(* Logix 5000 project; controller CLASE_1 Emulate 5570 rev 28.11; software revision 28.02; part 3 of 15 *)
(* tags used below, declared in another part *)
   Inp : BOOL;   // Alarm Condition Input 1=Alarm
   Cfg_Exists : BOOL;   // 1=Alarm configured to exist, 0=Does not exist, don't scan
   Cfg_ResetReqd : BOOL;   // 1=Latched Alarm, a Reset is required to clear this Alarm
   Cfg_AckReqd : BOOL;   // 1=Acknowledge required for this Alarm
   Cfg_AllowShelve : BOOL;   // 1=Allow Operator to Shelve this Alarm
   Cfg_AllowDisable : BOOL;   // 1=Allow Maintenance to Disable this Alarm
   Cfg_Severity : INT;   // Alarm Severity: 1..250=Low, 251..500=Medium, 501..750=High, 751..1000=Urgent
   Cfg_AlmMinOnT : DINT;   // Minimum time Alm output stays on (sec)
   Cfg_MaxShelfT : INT;   // Auto unshelve after shelved this long (1..32767 minutes)
   PCfg_AllowExist : BOOL;   // 1=Alarm can be configured to exist, 0=other configs make alarm meaningless
   PCmd_Ack : BOOL;   // Program Command to Acknowledge alarm
   PCmd_Suppress : BOOL;   // Program Command to Suppress by Design (inhibits new alarm)
   PCmd_Unsuppress : BOOL;   // Program Command to Unsuppress (allows new alarm)
   PCmd_Unshelve : BOOL;   // Program Command to Unshelve (e.g., on shift change)
   OCmd_Ack : BOOL;   // Operator Command to Acknowledge alarm
   OCmd_Shelve : BOOL;   // Operator Command to Shelve Alarm (inhibits new alarm)
   OCmd_Unshelve : BOOL;   // Operator Command to Unshelve alarm (allows new alarm)
   MCmd_Disable : BOOL;   // Maintenance Command to Disable alarm (inhibits new alarm)
   MCmd_Enable : BOOL;   // Maintenance Command to Enable alarm (allows new alarm)
   MCmd_Test : BOOL;   // Maintenance Command to Test alarm (issued for minimum alarm time)
   Val_MinToUnshelve : DINT;   // Number of minutes until this alarm unshelves itself (mmm:ss)
   Val_SecToUnshelve : DINT;   // Number of Seconds until this alarm unshelves itself (mmm:ss)
   Alm : ALIAS FOR Com_AE.0;   // Alarm output 1=In Alarm
   Ack : ALIAS FOR Com_AE.1;   // Alarm acknowledged status: 1=Ack rcvd
   Shelved : ALIAS FOR Com_AE.3;   // 1=Alarm has been Shelved by Operator (inhibits new alarm)
   Suppressed : ALIAS FOR Com_AE.6;   // 1=Alarm has been Suppressed by Program (inhibits new alarm)
   Disabled : ALIAS FOR Com_AE.9;   // 1=Alarm has been Disabled by Maintanance (inhibits new alarm)
   Err_Severity : BOOL;   // 1=Error in Config: Invalid Severity (use 1 to 4)
   Rdy_Ack : BOOL;   // Ready to receive OCmd_Ack (enables button)
   Rdy_Shelve : BOOL;   // Ready to receive OCmd_Shelve (enables button)
   Rdy_Unshelve : BOOL;   // Ready to receive OCmd_Unshelve (enables button)
   Rdy_Disable : BOOL;   // Ready to receive MCmd_Disable (enables button)
   Rdy_Enable : BOOL;   // Ready to receive MCmd_Enable (enables button)
   Rdy_Test : BOOL;   // Ready to receive MCmd_Test (enables button)
   P_Alarm : BOOL;   // Unique Parameter Name for auto - discovery
   Wrk_Alm : BOOL;   // Internal Alarm Status
   Wrk_Suppressed : BOOL;   // Internal Alarm Suppressed Status
   Wrk_AlmMinOnT : TIMER;   // Alarm output minimum ON time to be seen by alarm server
   Wrk_AutoAckT : TIMER;   // Time to clear Ack bit when Ack not required
   Wrk_ShelfT : TIMER;   // Time to auto Unshelve a Shelved Alarm
   Com_AE : INT;   // Communication with HMI / Alarm/Event Server (see bit descriptions)
   Cfg_Cond : STRING_20;   // Alarm Condition Text (e.g., "High-High PV")
   Wrk_SecToUnshelve : DINT;   // Number of seconds until this alarm unshelves itself
(* P_Alarm, continued *)

ROUTINE Logic   (* ladder *)
// Perform Alarm processing: delay, latch/reset, acknowledge, enable/disable, inhibit/uninhibit, suppress/unsuppress
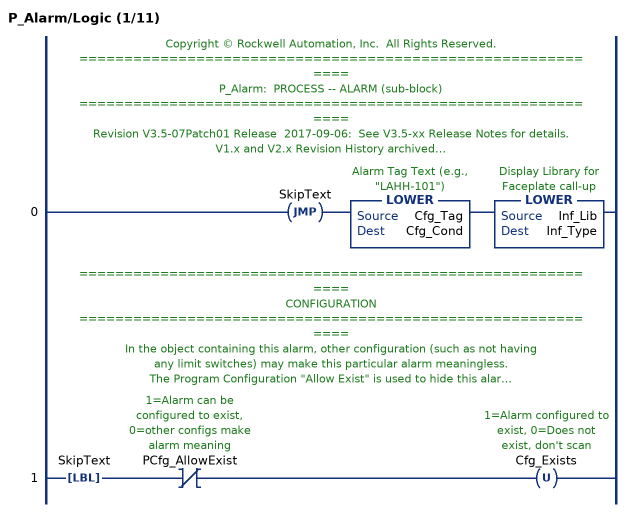
   // Copyright © Rockwell Automation, Inc.  All Rights Reserved.
   // ============================================================
   // P_Alarm:  PROCESS -- ALARM (sub-block)
   // ============================================================
   // Revision V3.5-07Patch01 Release  2017-09-06:  See V3.5-xx Release Notes for details.
   // V1.x and V2.x Revision History archived.
   // V3.0-00  2013-06-30:  Changed suppress to shelve, inhibit to suppress
   // (ANSI/ISA 18.2-2009 and FTView 7 alignment), added auto unshelve
   // timer, program command to unshelve.  Removed: Ack on shelve.
   // Added: clear Alm when Disabled, PCfg_AllowExist, Cfg_Tag,
   // Cfg_Cond, Inf_Lib, Inf_Type.  (Max Shelf Time is in MINUTES.)
   // Added local tag .Com_AE for FTAE communications.
   // V3.0-01  2013-07-30:  Changed range for Shelf Time to 1 to 34560 minutes.
   // V3.0-02  2013-10-30:  Changed Cfg_MaxShelfT check to LEQ 0.
   // (INT 1 to 32767 is valid.)
   // V3.1-00  2014-06-30:  Added Maintenace Test command, changed severity
   // ranges and names to match FTAE (for linking to FTView 8).
   // V3.1-01  2014-09-03:  Exposed shelf timer ACC/PRE (read-only).
   // V3.1-02  2014-09-30:  Modified FTAE interface for Disable/Enable and
   // Suppress/Unsuppress.  See "Alarm Setup" below!
   // V3.5-01  2016-01-29:  Fixed operation of Cfg_MaxShelfT, Cfg_AlmMinOnT.
   // V3.5-07Patch01  2017-09-06:  Modified for FTView ME "chattering alarm" ack timing.
   // ============================================================
   // This instruction monitors one input condition and provides one Alarm with:
   //   * configurable latching (reset required) and acknowledgement requirement
   //   * configurable alarm severity
   // 1..250 = Low  (blue, typ. informational)
   // 251-500 = Medium  (yelllow, typ. warning)
   // 501-750 = High  (red, typ. process exception)
   // 751-1000 = Urgent  (magenta, typ. equip. fault)
   // * configurable minimum ON time (e.g., to ensure it is seen by the HMI)
   // * commands to suppress/unsuppress (Prog), shelve/unshelve (Oper)
   // and disable/enable (Maint) the alarm.
   // * configurable amount of time shelved to automatically unshelve an alarm
   // * FTA&E support for suppressed, shelved and disabled states (V7.0)
   // NOTE regarding parameter naming:
   // FTA&E names (same as ALMD instruction) are used instead
   // of the ANSI/ISA 18.2-2009 names, as follows:
   // "Disabled" is the equivalent of "Out of Service" in ISA 18.2.
   // (the Disabled state is owned by Maintenance)
   // "Suppressed" is the equivalent of "Suppressed by Design" in ISA 18.2.
   // (the Suppressed state is owned by Program logic)
   // "Shelved" is the same as in ISA 18.2.
   // (the Shelved state is owned by Operator, but may be cleared
   // by Program logic based on time, shift change, etc.)
   // This instruction is usually nested within other instructions, with one instance
   // used for each Alarm generated by the containing instruction.  It may also be
   // used as a standalone instruction for Alarm conditions generated by custom logic.
   // ________________________________________
   // FTAE Alarm Setup:
   // ________________________________________
   // (object).(alarm).Com_AE.0:  Alarm to FTAE
   // .Com_AE.1:   Ack to/from FTAE
   // .Com_AE.3:   Shelved from FTAE Status
   // .Com_AE.4:   Shelve/Reshelve to FTAE Control (auto reset)
   // .Com_AE.5:   Unshelve to FTAE Control (auto reset)
   // .Com_AE.6:   Suppressed from FTAE Status
   // .Com_AE.7:   Suppress to FTAE Control (auto reset)
   // .Com_AE.8:   Unsuppress to FTAE Control (auto reset)
   // .Com_AE.9:   Disabled from FTAE Status
   // .Com_AE.10: Disable to FTAE Control (auto reset)
   // .Com_AE.11: Enable to FTAE Control (auto reset)
   // all other bits unused
   //     .Cfg_MaxShelfT is also used in FTAE config.
   // .Cfg_Severity is used by FTAE in FTView 8.x.
   // ============================================================
   // POWERUP / INVALID STATE HANDLING
   // ============================================================
   // All internal Work (state) bits maintain states through a power cycle and are
   // independent.  No first-scan logic is required.  See the Prescan routine for
   // powerup / prescan code.
   // ============================================================
   // SHOW LOCAL STRINGS
   // ============================================================
   // The STRINGs containing the text associated with each instance of this
   // instruction cannot be Input or Output Parameters, because STRINGs are not
   //  'atomic' types. (Inputs and Outputs must be SINT, INT, DINT, REAL, or BOOL.)
   // In order to make it easier to find and configure these STRINGs, this rung
   // was added.  THE JMP (and the LBL on the following rung)
   // MUST NOT BE REMOVED!!!
   // To view the STRINGs, go to the instruction instance (in LD or FBD), RIGHT-click
   // to bring up the context menu and select "Open Instruction Logic".
   // This rung will appear with the STRING values for the selected instance.
   // You may double-click the STRING values here to modify them as well.
   // #####  V3.0-00  2013-06-30:  Added rung; added new STRING local tags.  #####
   0: JMP(SkipText)LOWER(Cfg_Tag,Cfg_Cond)LOWER(Inf_Lib,Inf_Type);
   // ============================================================
   // CONFIGURATION
   // ============================================================
   // In the object containing this alarm, other configuration (such as not having
   // any limit switches) may make this particular alarm meaningless.
   // The Program Configuration "Allow Exist" is used to hide this alarm
   // on the object's faceplate and other graphics, and forces the Cfg_Exist to 0.
   // #####  V3.0-00 2013-06-30:  Added PCfg_AllowExist.  #####
   1: LBL(SkipText)XIO(PCfg_AllowExist)OTU(Cfg_Exists);
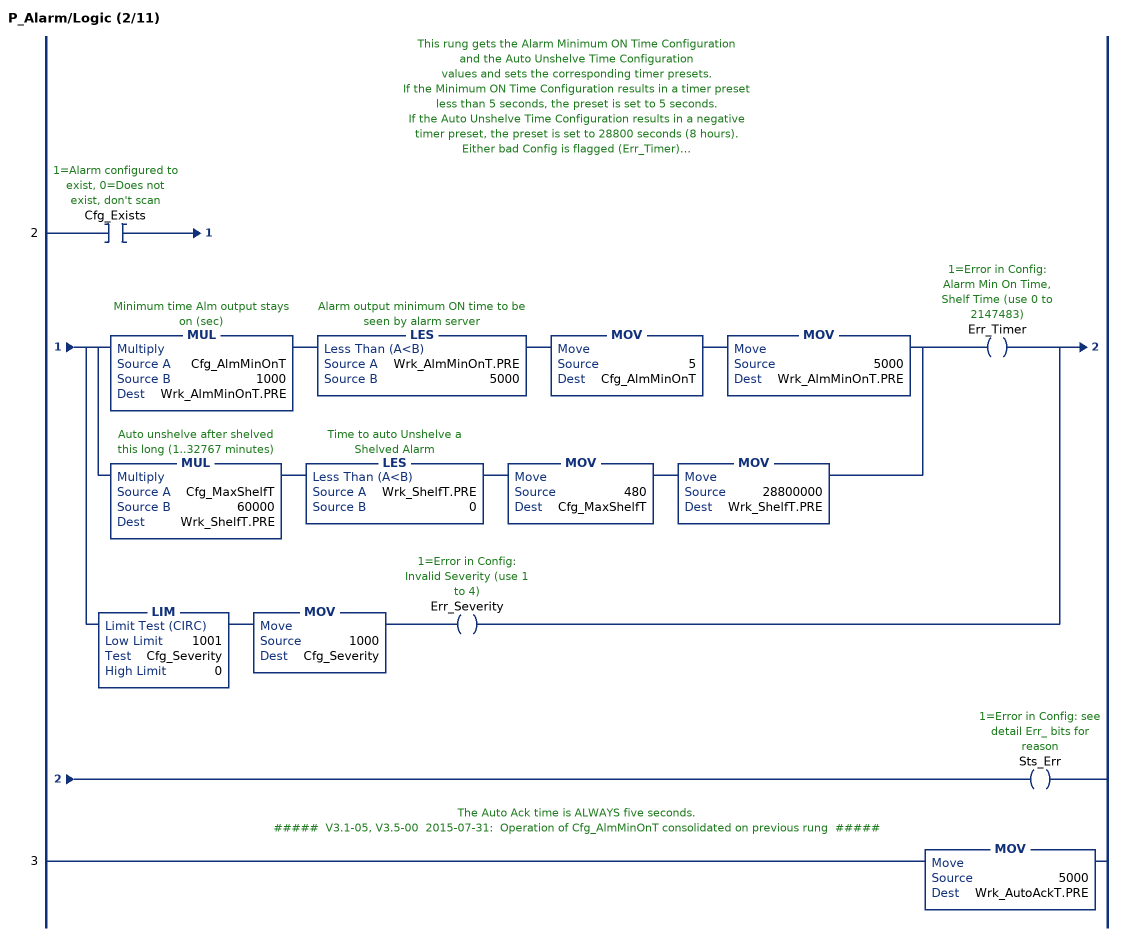
   // This rung gets the Alarm Minimum ON Time Configuration
   // and the Auto Unshelve Time Configuration
   // values and sets the corresponding timer presets.
   // If the Minimum ON Time Configuration results in a timer preset
   // less than 5 seconds, the preset is set to 5 seconds.
   // If the Auto Unshelve Time Configuration results in a negative
   // timer preset, the preset is set to 28800 seconds (8 hours).
   // Either bad Config is flagged (Err_Timer).
   // Bad Config is also flagged if the Cfg_Severity is out of range (valid = 1..1000) (Err_Severity).
   // #####  V3.0-00  2013-06-30:  Changed Program Inhibit to Suppress, Operator Suppress to Shelve.  #####
   // #####  Added Shelf Timer config check; if Severity out of range, make it "Fault".  #####
   // #####  V3.0-02  2013-10-30:  Changed Cfg_MaxShelfT check to LEQ 0.  (INT 1 to 32767 is valid.)  #####
   // #####  V3.1-05, V3.5-00  2015-07-31:  Fixed operation of Cfg_MaxShelfT = 0, Cfg_AlmMinOnT, rung comment.  #####
   2: XIC(Cfg_Exists)[[MUL(Cfg_AlmMinOnT,1000,Wrk_AlmMinOnT.PRE) LES(Wrk_AlmMinOnT.PRE,5000) MOV(5,Cfg_AlmMinOnT) MOV(5000,Wrk_AlmMinOnT.PRE) ,MUL(Cfg_MaxShelfT,60000,Wrk_ShelfT.PRE) LES(Wrk_ShelfT.PRE,0) MOV(480,Cfg_MaxShelfT) MOV(28800000,Wrk_ShelfT.PRE) ] OTE(Err_Timer) ,LIM(1001,Cfg_Severity,0) MOV(1000,Cfg_Severity) OTE(Err_Severity) ]OTE(Sts_Err);
   // The Auto Ack time is ALWAYS five seconds.
   // #####  V3.1-05, V3.5-00  2015-07-31:  Operation of Cfg_AlmMinOnT consolidated on previous rung  #####
   3: MOV(5000,Wrk_AutoAckT.PRE);
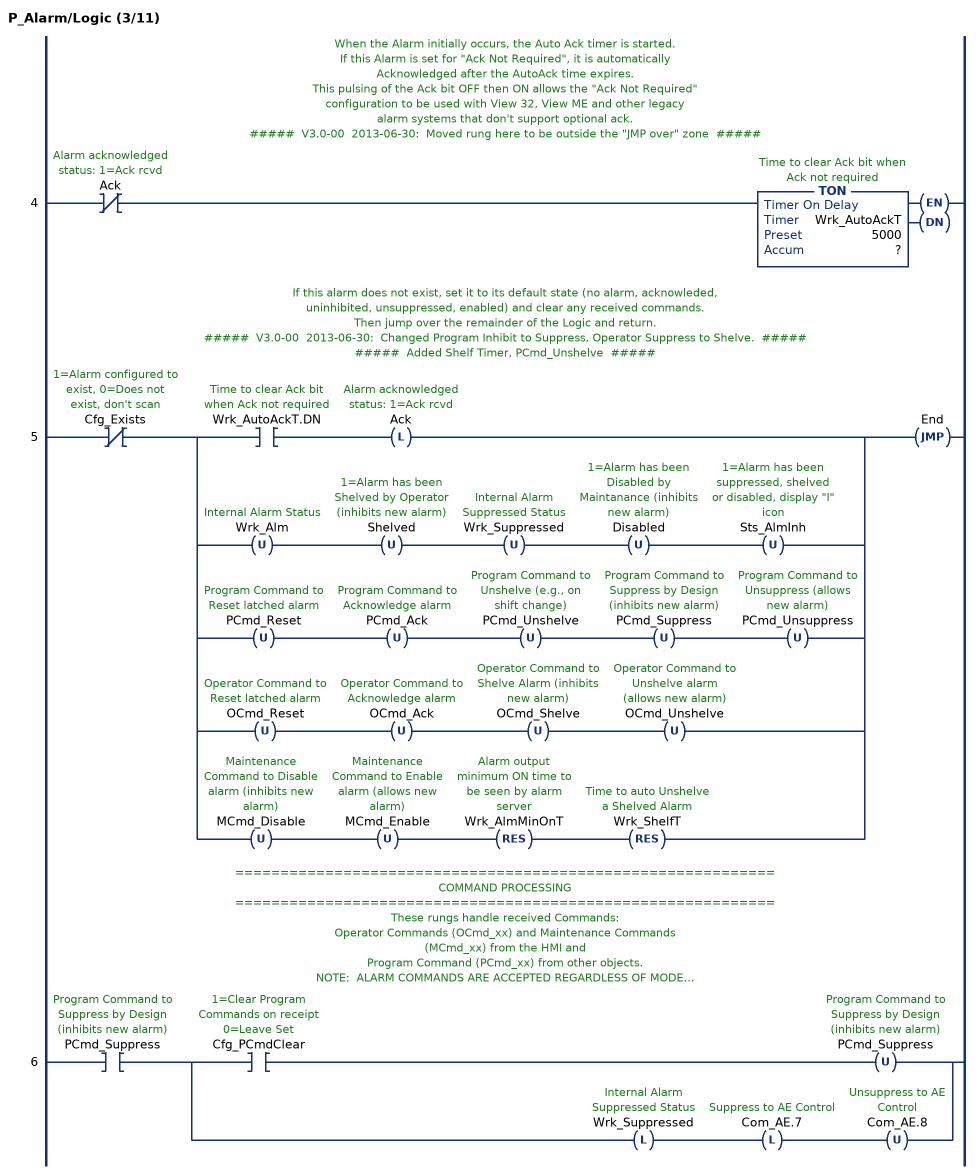
   // When the Alarm initially occurs, the Auto Ack timer is started.
   // If this Alarm is set for "Ack Not Required", it is automatically
   // Acknowledged after the AutoAck time expires.
   // This pulsing of the Ack bit OFF then ON allows the "Ack Not Required"
   // configuration to be used with View 32, View ME and other legacy
   // alarm systems that don't support optional ack.
   // #####  V3.0-00  2013-06-30:  Moved rung here to be outside the "JMP over" zone  #####
   4: XIO(Ack)TON(Wrk_AutoAckT,?,?);
   // If this alarm does not exist, set it to its default state (no alarm, acknowleded,
   // uninhibited, unsuppressed, enabled) and clear any received commands.
   // Then jump over the remainder of the Logic and return.
   // #####  V3.0-00  2013-06-30:  Changed Program Inhibit to Suppress, Operator Suppress to Shelve.  #####
   // #####  Added Shelf Timer, PCmd_Unshelve  #####
   5: XIO(Cfg_Exists)[XIC(Wrk_AutoAckT.DN) OTL(Ack) ,OTU(Wrk_Alm) OTU(Shelved) OTU(Wrk_Suppressed) OTU(Disabled) OTU(Sts_AlmInh) ,OTU(PCmd_Reset) OTU(PCmd_Ack) OTU(PCmd_Unshelve) OTU(PCmd_Suppress) OTU(PCmd_Unsuppress) ,OTU(OCmd_Reset) OTU(OCmd_Ack) OTU(OCmd_Shelve) OTU(OCmd_Unshelve) ,OTU(MCmd_Disable) OTU(MCmd_Enable) RES(Wrk_AlmMinOnT) RES(Wrk_ShelfT) ]JMP(End);
   // ============================================================
   // COMMAND PROCESSING
   // ============================================================
   // These rungs handle received Commands:
   // Operator Commands (OCmd_xx) and Maintenance Commands
   // (MCmd_xx) from the HMI and
   // Program Command (PCmd_xx) from other objects.
   // NOTE:  ALARM COMMANDS ARE ACCEPTED REGARDLESS OF MODE.
   // This rung receives the Program Alarm Inhibit Command.
   // If configured for EDGE, the Command is cleared.
   // #####  V3.1-02  2013-09-24:  Modified FTAE interface for Disable/Enable, Suppress/Unsuppress.  #####
   6: XIC(PCmd_Suppress)[XIC(Cfg_PCmdClear) OTU(PCmd_Suppress) ,OTL(Wrk_Suppressed) OTL(Com_AE.7) OTU(Com_AE.8) ];
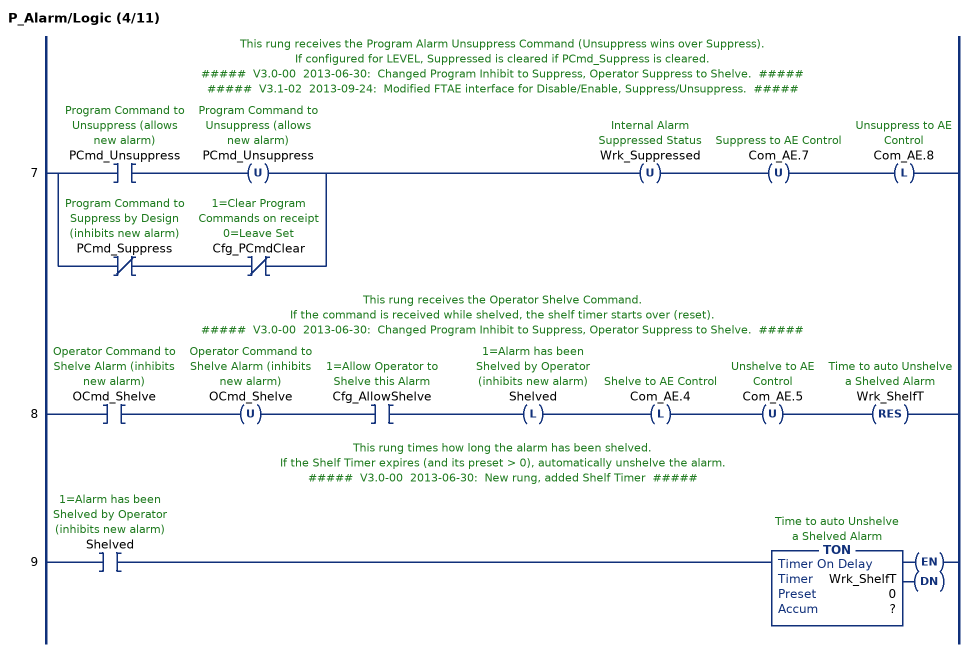
   // This rung receives the Program Alarm Unsuppress Command (Unsuppress wins over Suppress).
   // If configured for LEVEL, Suppressed is cleared if PCmd_Suppress is cleared.
   // #####  V3.0-00  2013-06-30:  Changed Program Inhibit to Suppress, Operator Suppress to Shelve.  #####
   // #####  V3.1-02  2013-09-24:  Modified FTAE interface for Disable/Enable, Suppress/Unsuppress.  #####
   7: [XIC(PCmd_Unsuppress) OTU(PCmd_Unsuppress) ,XIO(PCmd_Suppress) XIO(Cfg_PCmdClear) ]OTU(Wrk_Suppressed)OTU(Com_AE.7)OTL(Com_AE.8);
   // This rung receives the Operator Shelve Command.
   // If the command is received while shelved, the shelf timer starts over (reset).
   // #####  V3.0-00  2013-06-30:  Changed Program Inhibit to Suppress, Operator Suppress to Shelve.  #####
   8: XIC(OCmd_Shelve)OTU(OCmd_Shelve)XIC(Cfg_AllowShelve)OTL(Shelved)OTL(Com_AE.4)OTU(Com_AE.5)RES(Wrk_ShelfT);
   // This rung times how long the alarm has been shelved.
   // If the Shelf Timer expires (and its preset > 0), automatically unshelve the alarm.
   // #####  V3.0-00  2013-06-30:  New rung, added Shelf Timer  #####
   9: XIC(Shelved)TON(Wrk_ShelfT,?,?);
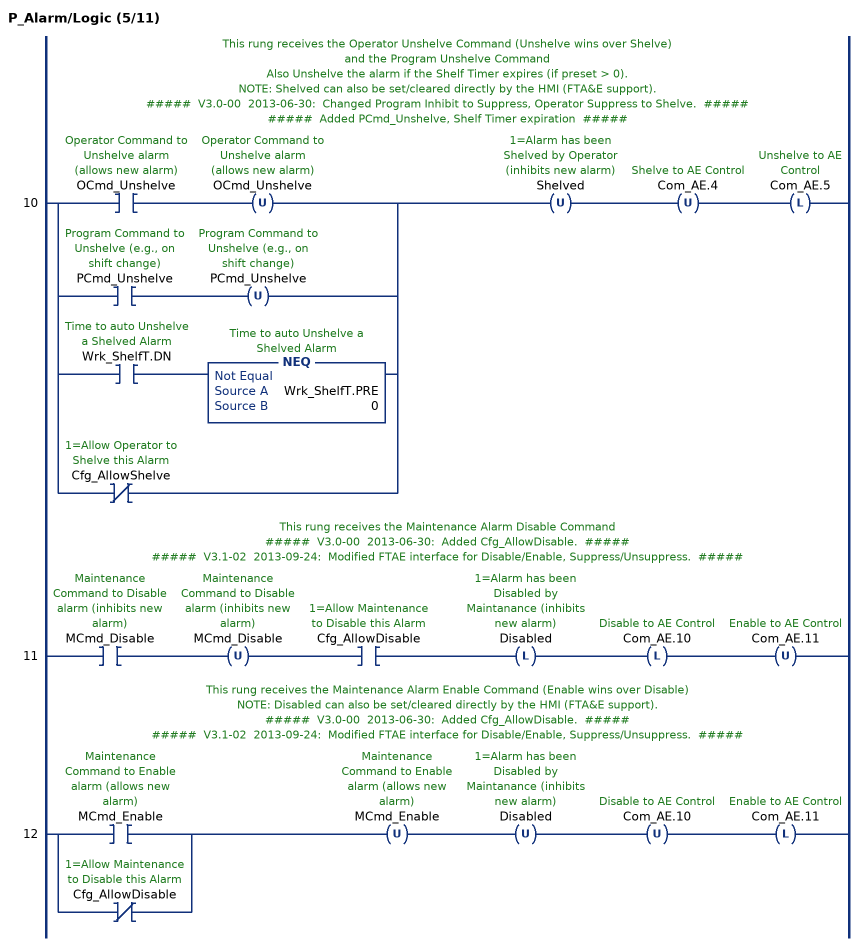
   // This rung receives the Operator Unshelve Command (Unshelve wins over Shelve)
   // and the Program Unshelve Command
   // Also Unshelve the alarm if the Shelf Timer expires (if preset > 0).
   // NOTE: Shelved can also be set/cleared directly by the HMI (FTA&E support).
   // #####  V3.0-00  2013-06-30:  Changed Program Inhibit to Suppress, Operator Suppress to Shelve.  #####
   // #####  Added PCmd_Unshelve, Shelf Timer expiration  #####
   10: [XIC(OCmd_Unshelve) OTU(OCmd_Unshelve) ,XIC(PCmd_Unshelve) OTU(PCmd_Unshelve) ,XIC(Wrk_ShelfT.DN) NEQ(Wrk_ShelfT.PRE,0) ,XIO(Cfg_AllowShelve) ]OTU(Shelved)OTU(Com_AE.4)OTL(Com_AE.5);
   // This rung receives the Maintenance Alarm Disable Command
   // #####  V3.0-00  2013-06-30:  Added Cfg_AllowDisable.  #####
   // #####  V3.1-02  2013-09-24:  Modified FTAE interface for Disable/Enable, Suppress/Unsuppress.  #####
   11: XIC(MCmd_Disable)OTU(MCmd_Disable)XIC(Cfg_AllowDisable)OTL(Disabled)OTL(Com_AE.10)OTU(Com_AE.11);
   // This rung receives the Maintenance Alarm Enable Command (Enable wins over Disable)
   // NOTE: Disabled can also be set/cleared directly by the HMI (FTA&E support).
   // #####  V3.0-00  2013-06-30:  Added Cfg_AllowDisable.  #####
   // #####  V3.1-02  2013-09-24:  Modified FTAE interface for Disable/Enable, Suppress/Unsuppress.  #####
   12: [XIC(MCmd_Enable) ,XIO(Cfg_AllowDisable) ]OTU(MCmd_Enable)OTU(Disabled)OTU(Com_AE.10)OTL(Com_AE.11);
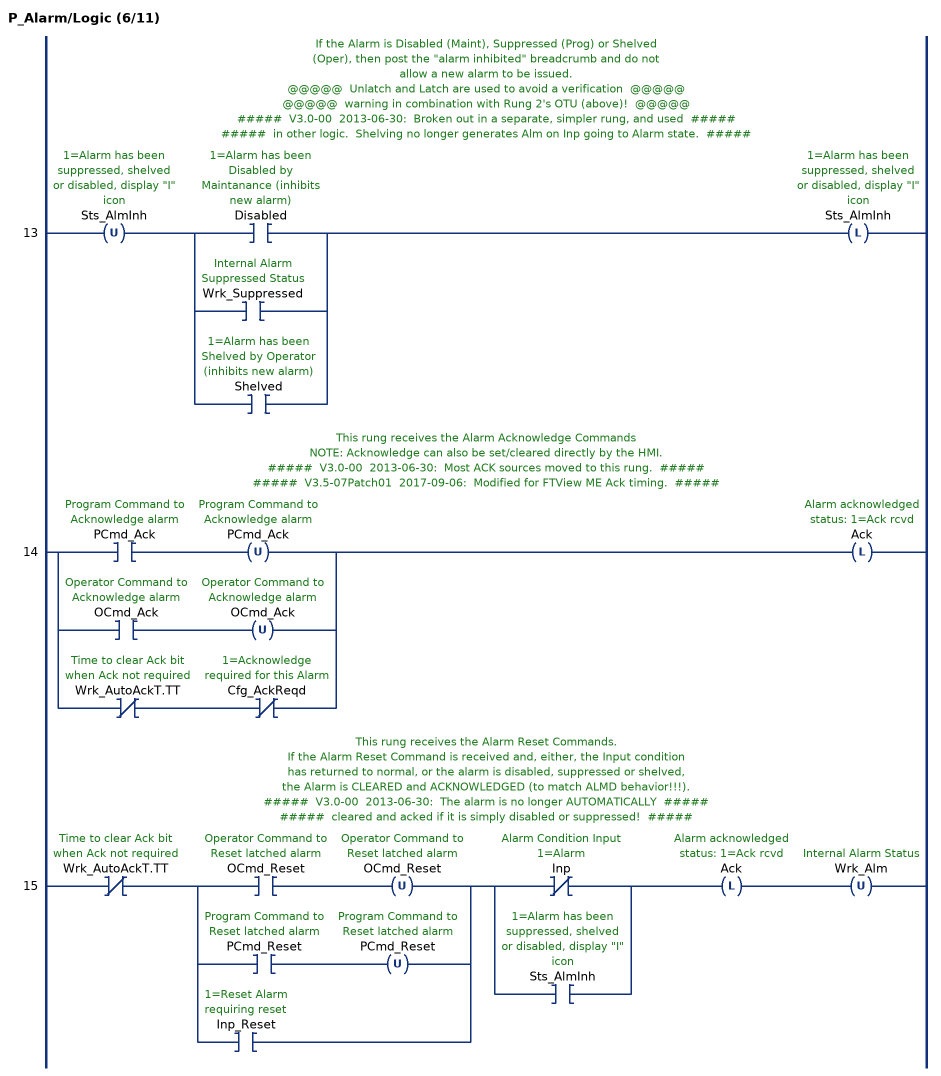
   // If the Alarm is Disabled (Maint), Suppressed (Prog) or Shelved
   // (Oper), then post the "alarm inhibited" breadcrumb and do not
   // allow a new alarm to be issued.
   // @@@@@  Unlatch and Latch are used to avoid a verification  @@@@@
   // @@@@@  warning in combination with Rung 2's OTU (above)!  @@@@@
   // #####  V3.0-00  2013-06-30:  Broken out in a separate, simpler rung, and used  #####
   // #####  in other logic.  Shelving no longer generates Alm on Inp going to Alarm state.  #####
   13: OTU(Sts_AlmInh)[XIC(Disabled) ,XIC(Wrk_Suppressed) ,XIC(Shelved) ]OTL(Sts_AlmInh);
   // This rung receives the Alarm Acknowledge Commands
   // NOTE: Acknowledge can also be set/cleared directly by the HMI.
   // #####  V3.0-00  2013-06-30:  Most ACK sources moved to this rung.  #####
   // #####  V3.5-07Patch01  2017-09-06:  Modified for FTView ME Ack timing.  #####
   14: [XIC(PCmd_Ack) OTU(PCmd_Ack) ,XIC(OCmd_Ack) OTU(OCmd_Ack) ,XIO(Wrk_AutoAckT.TT) XIO(Cfg_AckReqd) ]OTL(Ack);
   // This rung receives the Alarm Reset Commands.
   // If the Alarm Reset Command is received and, either, the Input condition
   // has returned to normal, or the alarm is disabled, suppressed or shelved,
   // the Alarm is CLEARED and ACKNOWLEDGED (to match ALMD behavior!!!).
   // #####  V3.0-00  2013-06-30:  The alarm is no longer AUTOMATICALLY  #####
   // #####  cleared and acked if it is simply disabled or suppressed!  #####
   15: XIO(Wrk_AutoAckT.TT)[XIC(OCmd_Reset) OTU(OCmd_Reset) ,XIC(PCmd_Reset) OTU(PCmd_Reset) ,XIC(Inp_Reset) ][XIO(Inp) ,XIC(Sts_AlmInh) ]OTL(Ack)OTU(Wrk_Alm);
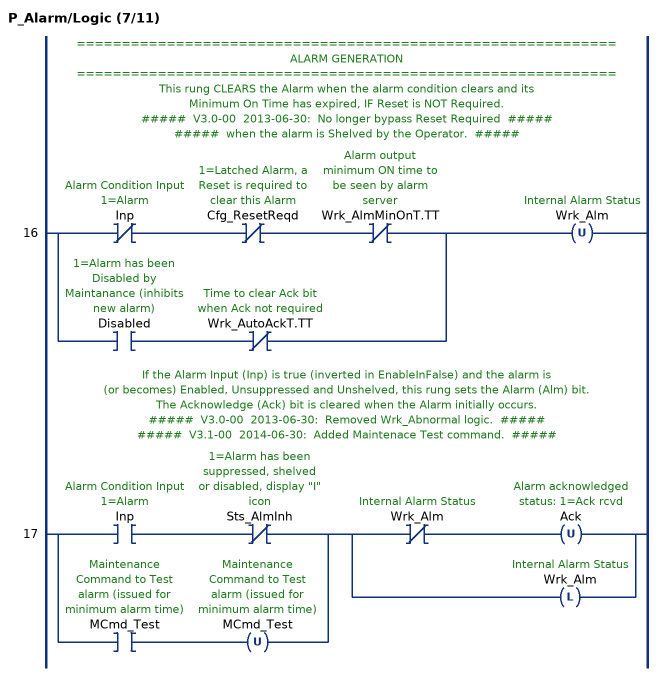
   // ============================================================
   // ALARM GENERATION
   // ============================================================
   // This rung CLEARS the Alarm when the alarm condition clears and its
   // Minimum On Time has expired, IF Reset is NOT Required.
   // #####  V3.0-00  2013-06-30:  No longer bypass Reset Required  #####
   // #####  when the alarm is Shelved by the Operator.  #####
   16: [XIO(Inp) XIO(Cfg_ResetReqd) XIO(Wrk_AlmMinOnT.TT) ,XIC(Disabled) XIO(Wrk_AutoAckT.TT) ]OTU(Wrk_Alm);
   // If the Alarm Input (Inp) is true (inverted in EnableInFalse) and the alarm is
   // (or becomes) Enabled, Unsuppressed and Unshelved, this rung sets the Alarm (Alm) bit.
   // The Acknowledge (Ack) bit is cleared when the Alarm initially occurs.
   // #####  V3.0-00  2013-06-30:  Removed Wrk_Abnormal logic.  #####
   // #####  V3.1-00  2014-06-30:  Added Maintenace Test command.  #####
   17: [XIC(Inp) XIO(Sts_AlmInh) ,XIC(MCmd_Test) OTU(MCmd_Test) ][XIO(Wrk_Alm) OTU(Ack) ,OTL(Wrk_Alm) ];
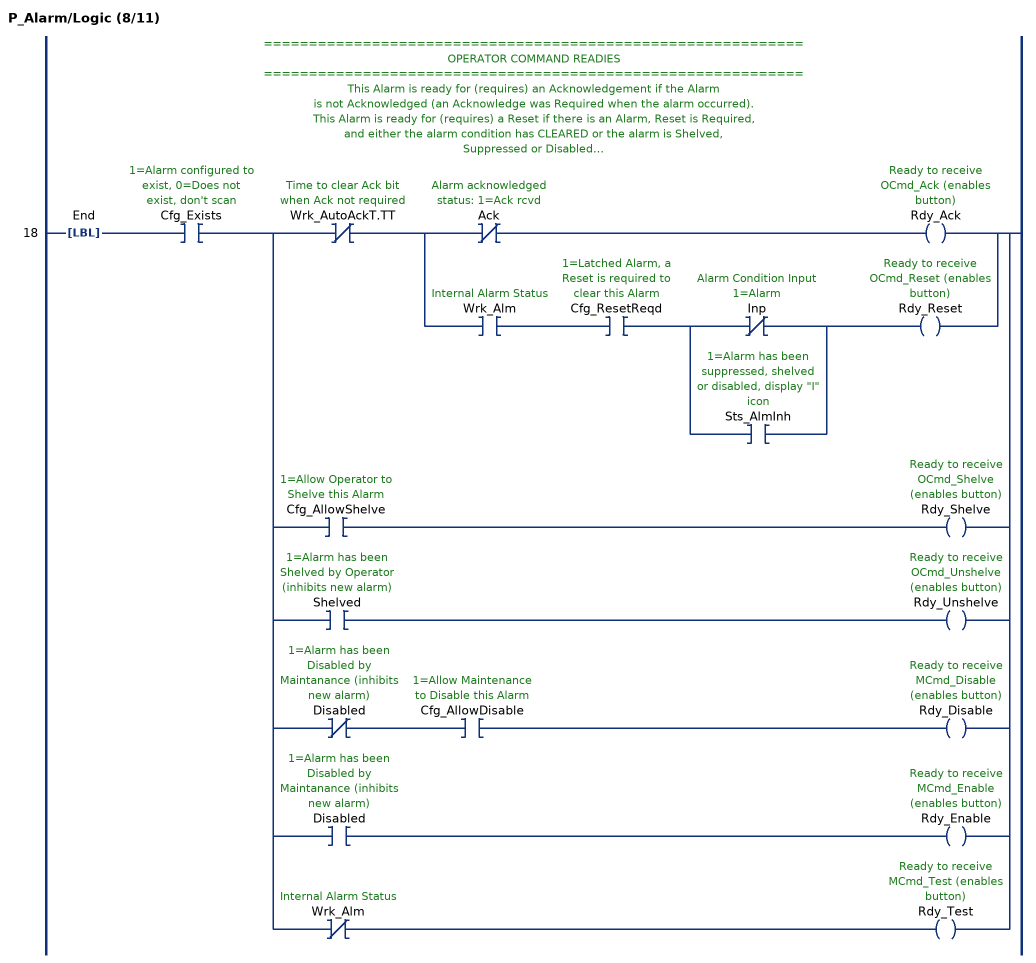
   // ============================================================
   // OPERATOR COMMAND READIES
   // ============================================================
   // This Alarm is ready for (requires) an Acknowledgement if the Alarm
   // is not Acknowledged (an Acknowledge was Required when the alarm occurred).
   // This Alarm is ready for (requires) a Reset if there is an Alarm, Reset is Required,
   // and either the alarm condition has CLEARED or the alarm is Shelved,
   // Suppressed or Disabled.
   // .
   // If the Alarm is NOT Shelved, it is ready for Shelve.
   // If the Alarm IS Shelved, it is ready for Unshelve.
   // If the Alarm is NOT Disabled, it is ready for Disable.
   // If the Alarm IS Disabled, it is ready for Enable.
   // NOTE: This rung appears before the Values/Status rung because the Rdy_Reset
   // condition is used to eliminate redundant logic in the rung below for Val_Notify.0.
   // #####  V3.0-00  2013-06-30:  Added sub-branch with Sts_AlmInh  #####
   // #####  V3.1-00  2014-06-30:  Added Maintenace Test command.  #####
   18: LBL(End)XIC(Cfg_Exists)[XIO(Wrk_AutoAckT.TT) [XIO(Ack) OTE(Rdy_Ack) ,XIC(Wrk_Alm) XIC(Cfg_ResetReqd) [XIO(Inp) ,XIC(Sts_AlmInh) ] OTE(Rdy_Reset) ] ,XIC(Cfg_AllowShelve) OTE(Rdy_Shelve) ,XIC(Shelved) OTE(Rdy_Unshelve) ,XIO(Disabled) XIC(Cfg_AllowDisable) OTE(Rdy_Disable) ,XIC(Disabled) OTE(Rdy_Enable) ,XIO(Wrk_Alm) OTE(Rdy_Test) ];
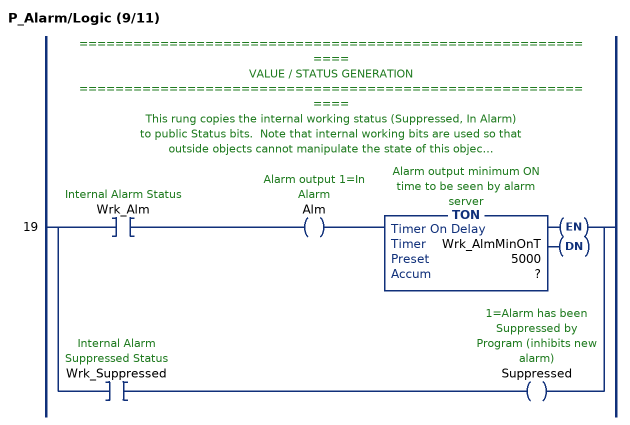
   // ============================================================
   // VALUE / STATUS GENERATION
   // ============================================================
   // This rung copies the internal working status (Suppressed, In Alarm)
   // to public Status bits.  Note that internal working bits are used so that
   // outside objects cannot manipulate the state of this object
   // by setting/clearing its Status and Alarm bits.
   // Public Status is generated for:
   // Alarm (with minimum ON time to be seen by polling)
   // Alarm Suppressed
   // Unsuppressed, Unshelved and Enabled are generated for HMI (FTVSE 7).
   // (Ack, Shelved and Disabled can be set/cleared by the HMI directly.
   // Note that these bits are "read/write" outputs in the parameter definition.)
   // #####  V3.0-00  2013-06-30:  New rung, some from below, new HMI bits.  #####
   19: [XIC(Wrk_Alm) OTE(Alm) TON(Wrk_AlmMinOnT,?,?) ,XIC(Wrk_Suppressed) OTE(Suppressed) ];
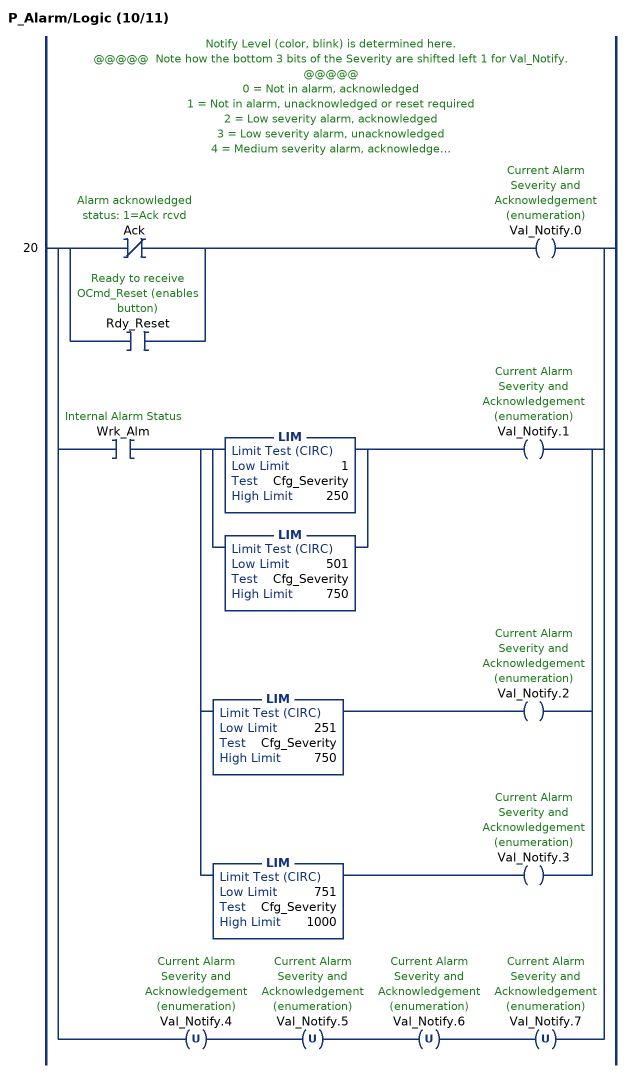
   // Notify Level (color, blink) is determined here.
   // @@@@@  Note how the bottom 3 bits of the Severity are shifted left 1 for Val_Notify.  @@@@@
   // 0 = Not in alarm, acknowledged
   // 1 = Not in alarm, unacknowledged or reset required
   // 2 = Low severity alarm, acknowledged
   // 3 = Low severity alarm, unacknowledged
   // 4 = Medium severity alarm, acknowledged
   // 5 = Medium severity alarm, unacknowledged
   // 6 = High severity alarm, acknowledged
   // 7 = High severity alarm, unacknowledged
   // 8 = Urgent severity alarm, acknowledged
   // 9 = Urgent severity alarm, unacknowledged
   // NOTE that the alarm bell icon will blink, even though the alarm is Acknowledged,
   // if an Alarm Reset is required (to get the Operator's attention).
   // #####  V3.0-00  2013-06-30:  Moved a few functions off this rung to logic above.  #####
   // #####  Names of Severity levels changed to Low, Medium, High, Highest  #####
   // #####  to match examples in ANSI/ISA-18.2-2009.  #####
   // #####  V3.1-00  2014-06-30:  Changed severity ranges, names to match FTAE  #####
   20: [[XIO(Ack) ,XIC(Rdy_Reset) ] OTE(Val_Notify.0) ,XIC(Wrk_Alm) [[LIM(1,Cfg_Severity,250) ,LIM(501,Cfg_Severity,750) ] OTE(Val_Notify.1) ,LIM(251,Cfg_Severity,750) OTE(Val_Notify.2) ,LIM(751,Cfg_Severity,1000) OTE(Val_Notify.3) ] ,OTU(Val_Notify.4) OTU(Val_Notify.5) OTU(Val_Notify.6) OTU(Val_Notify.7) ];
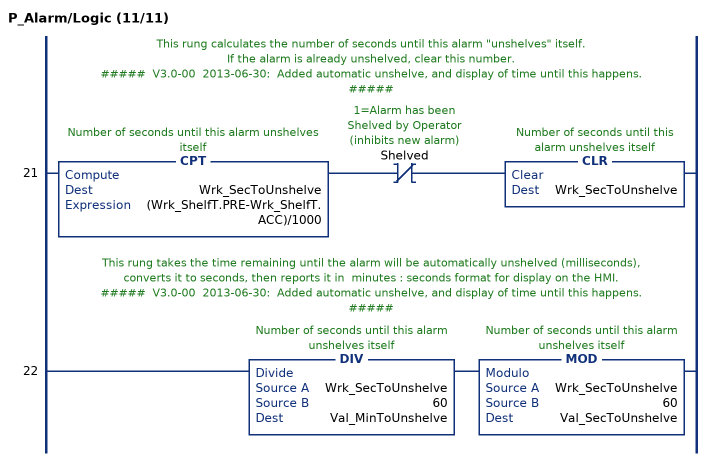
   // This rung calculates the number of seconds until this alarm "unshelves" itself.
   // If the alarm is already unshelved, clear this number.
   // #####  V3.0-00  2013-06-30:  Added automatic unshelve, and display of time until this happens.  #####
   21: CPT(Wrk_SecToUnshelve,(Wrk_ShelfT.PRE-Wrk_ShelfT.ACC)/1000)XIO(Shelved)CLR(Wrk_SecToUnshelve);
   // This rung takes the time remaining until the alarm will be automatically unshelved (milliseconds),
   // converts it to seconds, then reports it in  minutes : seconds format for display on the HMI.
   // #####  V3.0-00  2013-06-30:  Added automatic unshelve, and display of time until this happens.  #####
   22: DIV(Wrk_SecToUnshelve,60,Val_MinToUnshelve)MOD(Wrk_SecToUnshelve,60,Val_SecToUnshelve);
END_ROUTINE

ROUTINE Prescan   (* ladder *)
// Clear "lurking" Commands
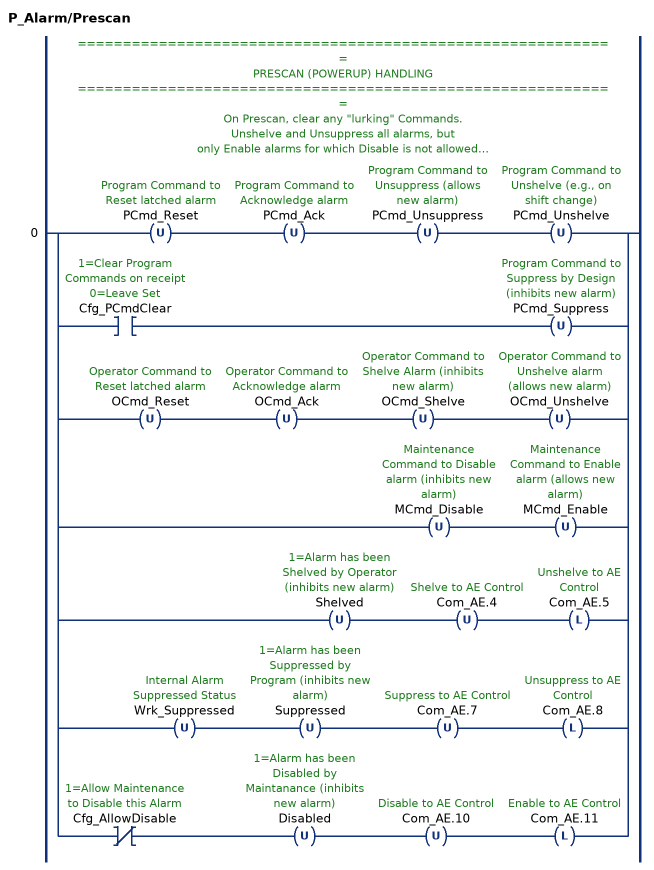
   // ============================================================
   // PRESCAN (POWERUP) HANDLING
   // ============================================================
   // On Prescan, clear any "lurking" Commands.
   // Unshelve and Unsuppress all alarms, but
   // only Enable alarms for which Disable is not allowed.
   // (Let Maintenance Disable persist through a power cycle...)
   // #####  V3.0-00  2013-06-30:  Added PCmd_Unshelve, AllowDisable, AllowShelve.  #####
   // #####  V3.1-02  2013-09-24:  Modified FTAE interface for Disable/Enable, Suppress/Unsuppress.  #####
   0: [OTU(PCmd_Reset) OTU(PCmd_Ack) OTU(PCmd_Unsuppress) OTU(PCmd_Unshelve) ,XIC(Cfg_PCmdClear) OTU(PCmd_Suppress) ,OTU(OCmd_Reset) OTU(OCmd_Ack) OTU(OCmd_Shelve) OTU(OCmd_Unshelve) ,OTU(MCmd_Disable) OTU(MCmd_Enable) ,OTU(Shelved) OTU(Com_AE.4) OTL(Com_AE.5) ,OTU(Wrk_Suppressed) OTU(Suppressed) OTU(Com_AE.7) OTL(Com_AE.8) ,XIO(Cfg_AllowDisable) OTU(Disabled) OTU(Com_AE.10) OTL(Com_AE.11) ];
END_ROUTINE
END_ADD_ON_INSTRUCTION

ADD_ON_INSTRUCTION P_DIn   (* revision 3.5 01 Release, vendor Rockwell Automation, ExecutePrescan, ExecuteEnableInFalse *)
// Discrete Input
// Revision note:
// See V3.5-xx Release Notes for details. Unchanged, using P_Alarm, P_Gate V3.5-01.
// Help:
// Copyright © Rockwell Automation, Inc.  All Rights Reserved.
// This instruction monitors a discrete (1 / 0) input and checks for alarm conditions.
// The Inp_Gate input must be set (=1, its default value) and the alarm enabled for
// the alarm (Alm) to occur.  The alarm will not occur until the Inp_Gate input has
// been set for the Gate Delay (Cfg_GateDly) time.  The Gate is used to enable the
// alarm when some other condition is true; for example, a high vibration switch should
// only generate an alarm when the associated motor has been running long enough
// to stabilize.
// The alarm is generated when the Inp_PV (process variable) input is different from
// the Inp_Target (target) input.  The Target indicates the "normal" condition.  For
// example, a flow switch should indicate flow when a pump is running and should
// not indicate flow when a pump is stopped.  The pump run status is used as the
// Target input, and when the switch does not match the target (within the allotted
// time), the Alarm (Flow Loss / Switch Failure) is generated.
// NOTE: the Inp_PV is inverted when the rung condition is false -- this allows the
// input to be a condition on the rung with P_DIn rather than mapped into Inp_PV.
// See P_DIn documentation for details.
// This instruction includes a substitute PV capability for a manually-entered state.
// This may be useful when a sensor is out for repair or for simulation and testing.
// Alarm is provided by a P_Alarm AOI instance.
// Status gating provided by P_Gate AOI instances.
VAR_INPUT
   Inp_PV : BOOL := 1; {visible}   // Input Signal (process variable) from Sensor
   Inp_PVBad : BOOL;   // Input Comm Status or Quality 1=Bad, 0=OK
   Inp_Target : BOOL := 1; {visible}   // Target State of Input (Disagree Status if not in Target State)
   Inp_Gate : ALIAS FOR TgtDisagreeGate.Inp_Gate; {visible}   // Gate Condition (=1 to enable Disagree Status)
   Inp_Sim : BOOL;   // 1=Use simulated PV (Set_SimPV); 0=Use Input (Inp_PV)
   Inp_Reset : BOOL;   // 1=Reset Alarm requiring reset
   Cfg_NoSubstPV : BOOL;   // 1=Disallow selection of Substitute PV
   Cfg_NormTextVis : BOOL := 1;   // 1=Display state text in "normal" state (= target), 0=hide (some HMI objects)
   Cfg_PCmdClear : BOOL := 1;   // 1=Clear Program Commands on receipt 0=Leave Set
   Cfg_HasTgtDisagreeAlm : ALIAS FOR TgtDisagree.Cfg_Exists;   // 1=Target Disagree Alarm exists and will be checked
   Cfg_TgtDisagreeResetReqd : ALIAS FOR TgtDisagree.Cfg_ResetReqd;   // 1=Target Disagree Alarm is latched in, requires Reset Command to clear
   Cfg_TgtDisagreeAckReqd : ALIAS FOR TgtDisagree.Cfg_AckReqd;   // 1=Target Disagree Alarm must be acknowledged
   Cfg_TgtDisagreeSeverity : ALIAS FOR TgtDisagree.Cfg_Severity;   // Target Disagree Alarm Severity: 1..250=Low, 251..500=Medium, 501..750=High, 751..1000=Urgent
   Cfg_GateDly : ALIAS FOR TgtDisagreeGate.Cfg_GateDly;   // Time Inp_Gate must be true before Disagree Status is checked (sec)
   Cfg_Debounce : REAL;   // Minimum time Input Sts must maintain state (sec)
   Cfg_TgtDisagreeOnDly : ALIAS FOR TgtDisagreeGate.Cfg_OnDly;   // Minimum time for Input to disagree with Target to raise Status (sec)
   Cfg_TgtDisagreeOffDly : ALIAS FOR TgtDisagreeGate.Cfg_OffDly;   // Minimum time for Input to agree with Target to clear Status (sec)
   MSet_SubstPV : BOOL;   // Maintenance-Entered Substitute PV
   Set_SimPV : BOOL;   // PV used in Simulation (Inp_Sim=1)
   PCmd_Reset : BOOL;   // Program Command to Reset all latched Alarms
   PCmd_TgtDisagreeAck : ALIAS FOR TgtDisagree.PCmd_Ack;   // Program Command to Acknowledge the Target Disagree Alarm
   PCmd_TgtDisagreeSuppress : ALIAS FOR TgtDisagree.PCmd_Suppress;   // Program Command to Suppress the Target Disagree Alarm
   PCmd_TgtDisagreeUnsuppress : ALIAS FOR TgtDisagree.PCmd_Unsuppress;   // Program Command to Unsuppress the Target Disagree Alarm
   PCmd_TgtDisagreeUnshelve : ALIAS FOR TgtDisagree.PCmd_Unshelve;   // Program Command to Unshelve the Target Disagree Alarm
   MCmd_SubstPV : BOOL;   // Maintenance Command to use Substitute PV (override input)
   MCmd_InpPV : BOOL;   // Maintenance Command to use Input PV (normal)
   OCmd_Reset : BOOL;   // Operator Command to Reset all latched Alarms
   OCmd_ResetAckAll : BOOL;   // Operator Command to Reset and Acknowledge all Alarms
END_VAR
VAR_OUTPUT
   SrcQ_IO : SINT; {access Read Only}   // Source and Quality of primary I/O (enumeration)
   SrcQ : SINT; {access Read Only}   // Source and Quality of primary Val/Sts (enumeration)
   Val_Sts : SINT; {access Read Only}   // Device Confirmed Sts 0=PV Good, 6=PV Bad, 7=Substitute PV
   Val_Fault : SINT; {access Read Only}   // Device Fault Status 0=none, 16=Tgt Disagree, 34=CfgErr
   Val_Notify : SINT; {access Read Only}   // Current Alarm Level and Acknowledgement (enumeration)
   Sts : BOOL; {access Read Only, visible}   // Discrete Input Status (incl. Debounce, Manual Override, if used)
   Sts_PV : BOOL; {access Read Only, visible}   // Discrete Input Status (actual, not subject to Override)
   Sts_SubstPV : BOOL; {access Read Only}   // 1=Using Substitute PV (Input being overridden)
   Sts_InpPV : BOOL; {access Read Only}   // 1=Using Input PV (normal)
   Sts_PVBad : BOOL; {access Read Only}   // Input Comm Status/ Quality (0=OK, 1=Bad)
   Sts_MaintByp : BOOL; {access Read Only}   // 1=Device has a Maintenance Bypass function active
   Sts_AlmInh : BOOL; {access Read Only}   // 1=One or more Alarms Shelved, Disabled or Suppressed
   Sts_Err : BOOL; {access Read Only, visible}   // 1=Error in Config: see detail bits for reason
   Err_Timer : BOOL; {access Read Only}   // 1=Error in Config: Invalid Timer Preset (use 0 to 2147483)
   Err_Alarm : BOOL; {access Read Only}   // 1=Error in Config: Alarm Min On Time, Shelf Time, Severity
   Sts_TgtDisagreeCmp : ALIAS FOR TgtDisagreeGate.Inp;   // Input vs. Target comparicon result 1=Disagree
   Sts_TgtDisagreeGate : ALIAS FOR TgtDisagreeGate.Sts_Gate; {access Read Only}   // Target Disagree Gate Delay Status, 1=done
   Sts_TgtDisagree : ALIAS FOR TgtDisagree.Inp;   // 1=Input is not in Target state
   Alm_TgtDisagree : ALIAS FOR TgtDisagree.Alm;   // 1=Alarm: Input is not in Target state
   Ack_TgtDisagree : ALIAS FOR TgtDisagree.Ack;   // 1=Target Disagree Alarm has been acknowledged
   Sts_TgtDisagreeDisabled : ALIAS FOR TgtDisagree.Disabled;   // 1=Target Disagree Alarm has been Disabled by Maintenance
   Sts_TgtDisagreeShelved : ALIAS FOR TgtDisagree.Shelved;   // 1=Target Disagree Alarm has been Shelved by Operator
   Sts_TgtDisagreeSuppressed : ALIAS FOR TgtDisagree.Suppressed;   // 1=Target Disagree Alarm has been Suppressed by Program
   Rdy_SubstPV : BOOL; {access Read Only}   // 1=Ready for MCmd_SubstPV
   Rdy_InpPV : BOOL; {access Read Only}   // 1=Ready for MCmd_InpPV
   Rdy_Reset : BOOL; {access Read Only}   // 1=At least one Alarm requires Reset
   Rdy_ResetAckAll : BOOL; {access Read Only}   // 1=At least one Alarm requires Acknowledgement
   P_DIn : BOOL;   // Unique Parameter Name for auto - discovery
END_VAR
VAR
   Cfg_Tag : STRING_20 := 'P_DIn';   // Tagname for display on HMI
   Cfg_Desc : STRING_40 := 'Discrete Input';   // Description for display on HMI
   Cfg_Label : STRING_20 := 'Discrete Input';   // Label for graphic symbol displayed on HMI
   Wrk_Sts : BOOL; {access None}   // Internal Status (after Manual Override selection)
   TgtDisagree : P_Alarm := (Cfg_AckReqd := 1, Cfg_AllowShelve := 1, Cfg_AllowDisable := 1, Cfg_PCmdClear := 1, Cfg_Severity := 750, Cfg_AlmMinOnT := 5, PCfg_AllowExist := 1, Ack := 1);   // Target Disagree Alarm
   Wrk_FallT : TIMER; {access None}   // Timer to ensure Status LOW time on falling edge
   Wrk_RiseT : TIMER; {access None}   // Timer to ensure Status HIGH time on rising edge
   Wrk_SubstPV : BOOL; {access None}   // Internal flag: Using Substitute PV
   Cfg_1StText : STRING_8 := 'On';   // Text to display in PV=1 State
   Cfg_0StText : STRING_8 := 'Off';   // Text to display in PV=0 State
   Inf_Tab : SINT;   // Tab to display (FTView ME)
   Wrk_Fault : SINT; {access None}   // Buffer for building Val_Fault
   Wrk_Status : SINT; {access None}   // Buffer for building Val_Sts
   Wrk_SrcQ : SINT; {access None}   // Register for building Source / Quality enumeration
   Inf_Type : STRING_16 := 'P_DIn'; {access Read Only}   // Must contain AOI name, used for HMI and Information S/W
   TgtDisagreeGate : P_Gate := (Inp_Gate := 1);   // Target Disagree Condition Gate/Delay
   Inf_Lib : STRING_12 := 'RA-BAS'; {access Read Only}   // Display Library for Faceplate call-up
END_VAR

ROUTINE EnableInFalse   (* ladder *)
// Same as main Logic routine, except Inp is inverted (for use in LD logic)
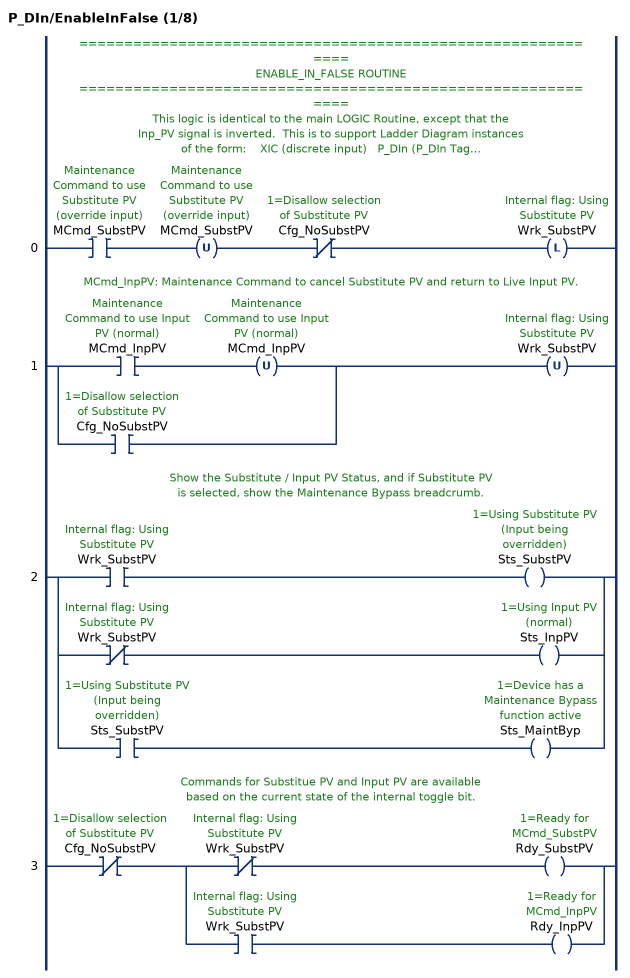
   // ============================================================
   // ENABLE_IN_FALSE ROUTINE
   // ============================================================
   // This logic is identical to the main LOGIC Routine, except that the
   // Inp_PV signal is inverted.  This is to support Ladder Diagram instances
   // of the form:    XIC (discrete input)   P_DIn (P_DIn Tag)
   // ============================================================
   // POWERUP / INVALID STATE HANDLING
   // ============================================================
   // All internal Work (state) bits maintain states through a power cycle and are
   // independent.  No Powerup / Invalid State Handling logic is required.
   // ============================================================
   // COMMAND PROCESSING
   // ============================================================
   // These rungs handle received Commands:
   // NOTE:  Operator Commands for P_Alarm are sent directly to the contained AOI.
   // MCmd_SubstPV: Maintenance Command to select Maintenance-entered substitute PV
   // Do not allow this Command if Cfg_NoSubstPV is set.
   0: XIC(MCmd_SubstPV)OTU(MCmd_SubstPV)XIO(Cfg_NoSubstPV)OTL(Wrk_SubstPV);
   // MCmd_InpPV: Maintenance Command to cancel Substitute PV and return to Live Input PV.
   1: [XIC(MCmd_InpPV) OTU(MCmd_InpPV) ,XIC(Cfg_NoSubstPV) ]OTU(Wrk_SubstPV);
   // Show the Substitute / Input PV Status, and if Substitute PV
   // is selected, show the Maintenance Bypass breadcrumb.
   2: [XIC(Wrk_SubstPV) OTE(Sts_SubstPV) ,XIO(Wrk_SubstPV) OTE(Sts_InpPV) ,XIC(Sts_SubstPV) OTE(Sts_MaintByp) ];
   // Commands for Substitue PV and Input PV are available
   // based on the current state of the internal toggle bit.
   3: XIO(Cfg_NoSubstPV)[XIO(Wrk_SubstPV) OTE(Rdy_SubstPV) ,XIC(Wrk_SubstPV) OTE(Rdy_InpPV) ];
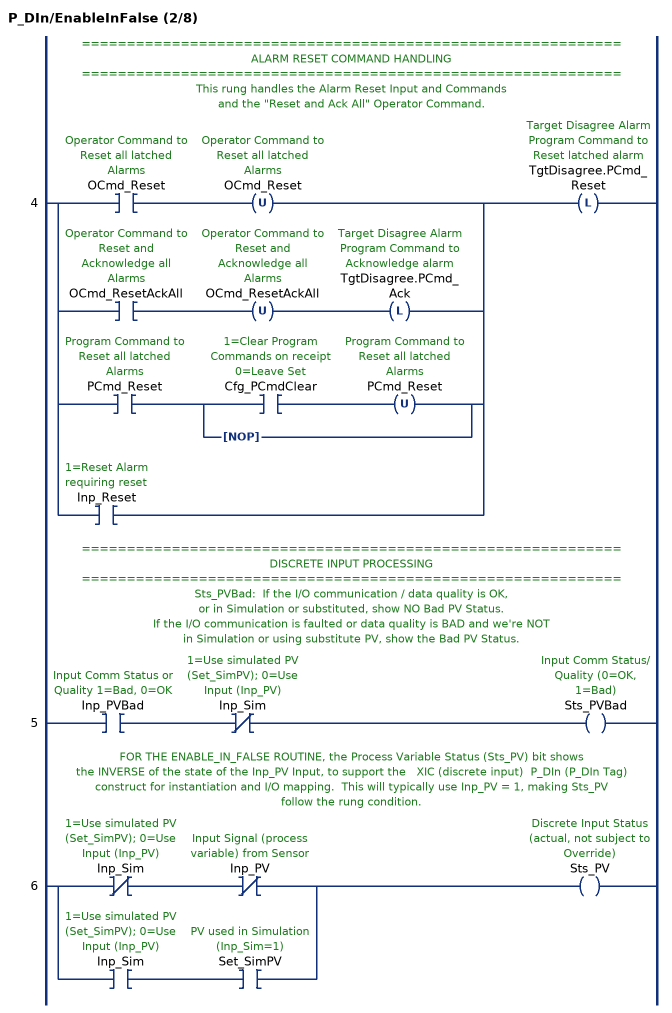
   // ============================================================
   // ALARM RESET COMMAND HANDLING
   // ============================================================
   // This rung handles the Alarm Reset Input and Commands
   // and the "Reset and Ack All" Operator Command.
   4: [XIC(OCmd_Reset) OTU(OCmd_Reset) ,XIC(OCmd_ResetAckAll) OTU(OCmd_ResetAckAll) OTL(TgtDisagree.PCmd_Ack) ,XIC(PCmd_Reset) [XIC(Cfg_PCmdClear) OTU(PCmd_Reset) ,NOP() ] ,XIC(Inp_Reset) ]OTL(TgtDisagree.PCmd_Reset);
   // ============================================================
   // DISCRETE INPUT PROCESSING
   // ============================================================
   // Sts_PVBad:  If the I/O communication / data quality is OK,
   // or in Simulation or substituted, show NO Bad PV Status.
   // If the I/O communication is faulted or data quality is BAD and we're NOT
   // in Simulation or using substitute PV, show the Bad PV Status.
   5: XIC(Inp_PVBad)XIO(Inp_Sim)OTE(Sts_PVBad);
   // FOR THE ENABLE_IN_FALSE ROUTINE, the Process Variable Status (Sts_PV) bit shows
   // the INVERSE of the state of the Inp_PV Input, to support the   XIC (discrete input)  P_DIn (P_DIn Tag)
   // construct for instantiation and I/O mapping.  This will typically use Inp_PV = 1, making Sts_PV
   // follow the rung condition.
   6: [XIO(Inp_Sim) XIO(Inp_PV) ,XIC(Inp_Sim) XIC(Set_SimPV) ]OTE(Sts_PV);
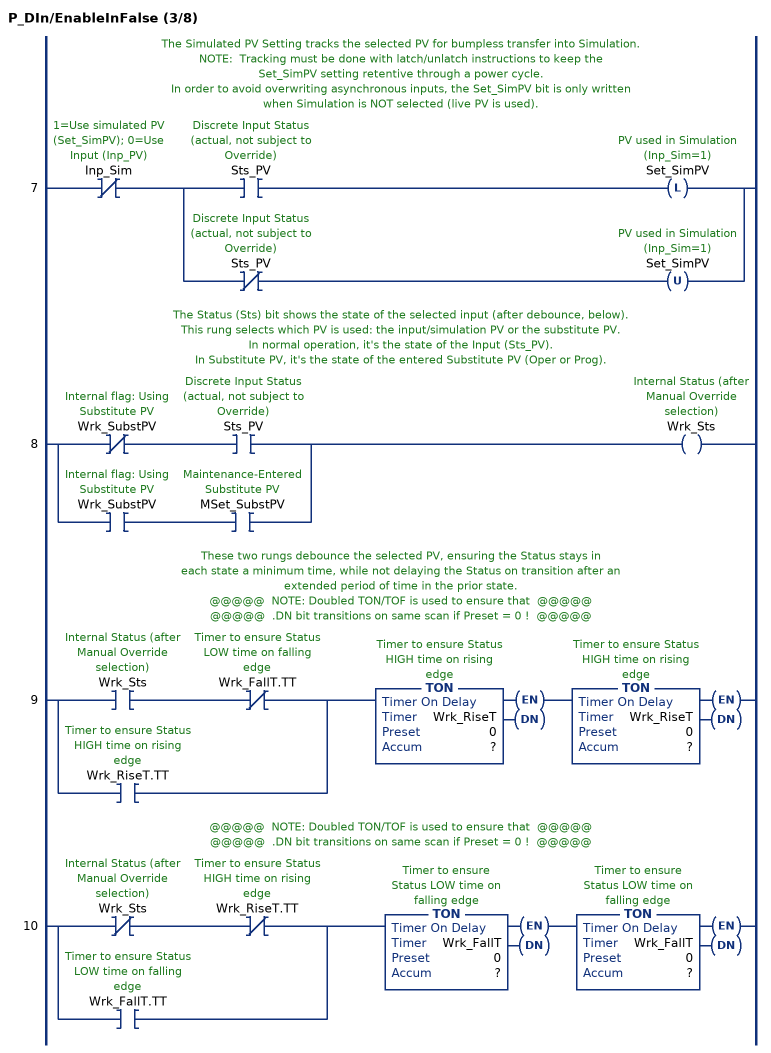
   // The Simulated PV Setting tracks the selected PV for bumpless transfer into Simulation.
   // NOTE:  Tracking must be done with latch/unlatch instructions to keep the
   // Set_SimPV setting retentive through a power cycle.
   // In order to avoid overwriting asynchronous inputs, the Set_SimPV bit is only written
   // when Simulation is NOT selected (live PV is used).
   7: XIO(Inp_Sim)[XIC(Sts_PV) OTL(Set_SimPV) ,XIO(Sts_PV) OTU(Set_SimPV) ];
   // The Status (Sts) bit shows the state of the selected input (after debounce, below).
   // This rung selects which PV is used: the input/simulation PV or the substitute PV.
   // In normal operation, it's the state of the Input (Sts_PV).
   // In Substitute PV, it's the state of the entered Substitute PV (Oper or Prog).
   8: [XIO(Wrk_SubstPV) XIC(Sts_PV) ,XIC(Wrk_SubstPV) XIC(MSet_SubstPV) ]OTE(Wrk_Sts);
   // These two rungs debounce the selected PV, ensuring the Status stays in
   // each state a minimum time, while not delaying the Status on transition after an
   // extended period of time in the prior state.
   // @@@@@  NOTE: Doubled TON/TOF is used to ensure that  @@@@@
   // @@@@@  .DN bit transitions on same scan if Preset = 0 !  @@@@@
   9: [XIC(Wrk_Sts) XIO(Wrk_FallT.TT) ,XIC(Wrk_RiseT.TT) ]TON(Wrk_RiseT,?,?)TON(Wrk_RiseT,?,?);
   // @@@@@  NOTE: Doubled TON/TOF is used to ensure that  @@@@@
   // @@@@@  .DN bit transitions on same scan if Preset = 0 !  @@@@@
   10: [XIO(Wrk_Sts) XIO(Wrk_RiseT.TT) ,XIC(Wrk_FallT.TT) ]TON(Wrk_FallT,?,?)TON(Wrk_FallT,?,?);
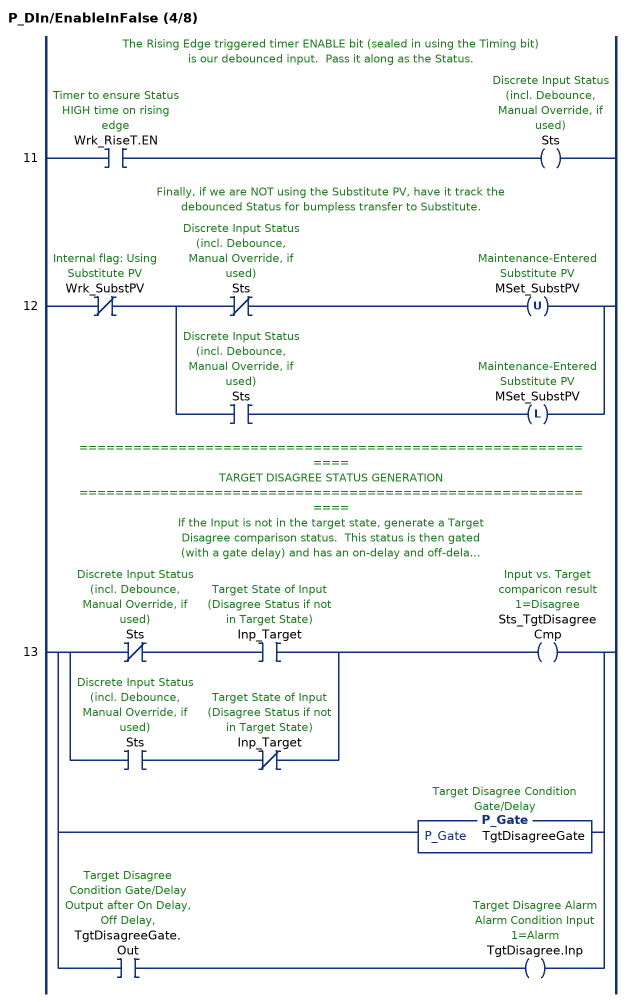
   // The Rising Edge triggered timer ENABLE bit (sealed in using the Timing bit)
   // is our debounced input.  Pass it along as the Status.
   11: XIC(Wrk_RiseT.EN)OTE(Sts);
   // Finally, if we are NOT using the Substitute PV, have it track the
   // debounced Status for bumpless transfer to Substitute.
   12: XIO(Wrk_SubstPV)[XIO(Sts) OTU(MSet_SubstPV) ,XIC(Sts) OTL(MSet_SubstPV) ];
   // ============================================================
   // TARGET DISAGREE STATUS GENERATION
   // ============================================================
   // If the Input is not in the target state, generate a Target
   // Disagree comparison status.  This status is then gated
   // (with a gate delay) and has an on-delay and off-delay
   // before feeding the final Target Disagree status bit.
   // #####  V3.0-00  2013-06-30:  Using P_Gate 3.0  #####
   13: [[XIO(Sts) XIC(Inp_Target) ,XIC(Sts) XIO(Inp_Target) ] OTE(Sts_TgtDisagreeCmp) ,P_Gate(TgtDisagreeGate) ,XIC(TgtDisagreeGate.Out) OTE(TgtDisagree.Inp) ];
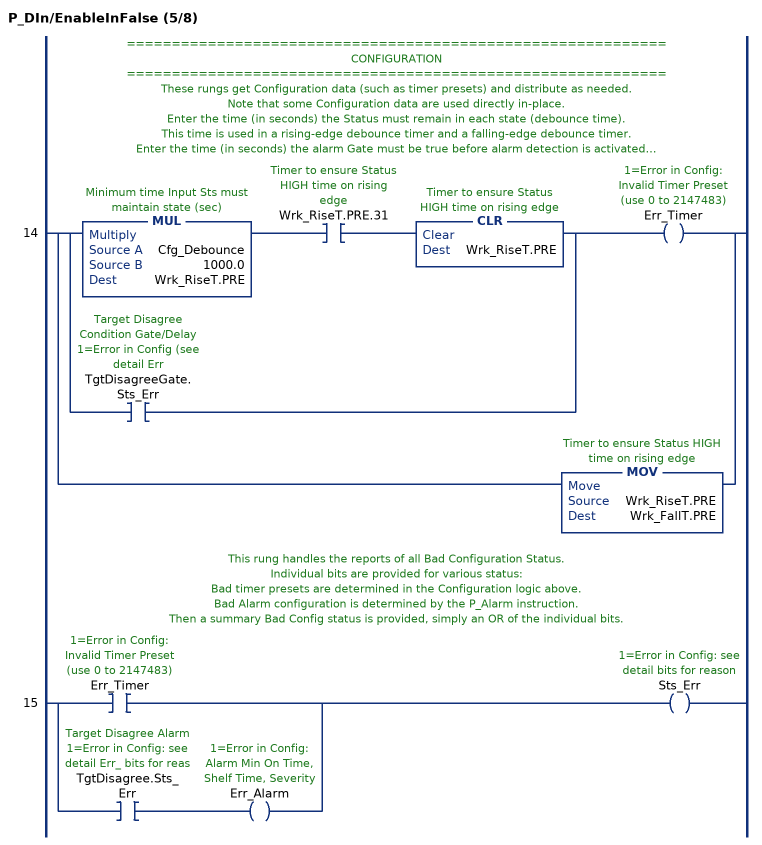
   // ============================================================
   // CONFIGURATION
   // ============================================================
   // These rungs get Configuration data (such as timer presets) and distribute as needed.
   // Note that some Configuration data are used directly in-place.
   // Enter the time (in seconds) the Status must remain in each state (debounce time).
   // This time is used in a rising-edge debounce timer and a falling-edge debounce timer.
   // Enter the time (in seconds) the alarm Gate must be true before alarm detection is activated.
   // Enter the On-Delay and Off-Delay times (in seconds) for the Target Disagree Status
   // (which feeds the Target Disagree Alarm).
   // If the timer preset calcuated wraps negative (more than 2.14... million seconds), then establish
   // a valid limit value for the Preset.  Note that a negative timer preset will fault the controller!!!
   // #####  V3.0-00  2013-06-30:  Using P_Gate 3.0  #####
   14: [[MUL(Cfg_Debounce,1000.0,Wrk_RiseT.PRE) XIC(Wrk_RiseT.PRE.31) CLR(Wrk_RiseT.PRE) ,XIC(TgtDisagreeGate.Sts_Err) ] OTE(Err_Timer) ,MOV(Wrk_RiseT.PRE,Wrk_FallT.PRE) ];
   // This rung handles the reports of all Bad Configuration Status.
   // Individual bits are provided for various status:
   // Bad timer presets are determined in the Configuration logic above.
   // Bad Alarm configuration is determined by the P_Alarm instruction.
   // Then a summary Bad Config status is provided, simply an OR of the individual bits.
   15: [XIC(Err_Timer) ,XIC(TgtDisagree.Sts_Err) OTE(Err_Alarm) ]OTE(Sts_Err);
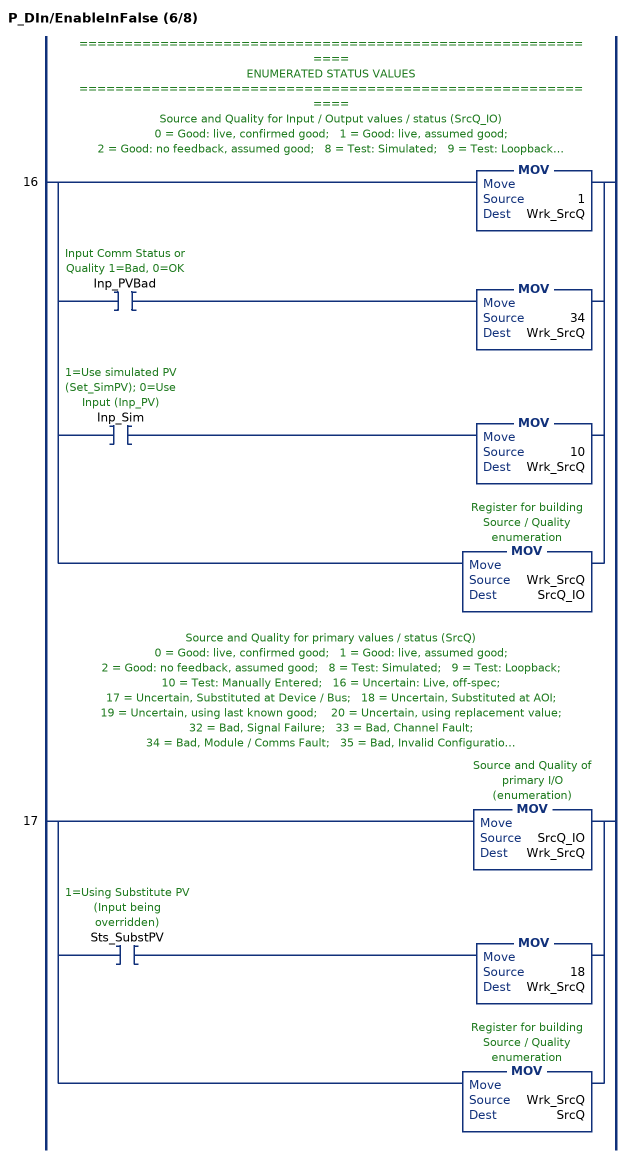
   // ============================================================
   // ENUMERATED STATUS VALUES
   // ============================================================
   // Source and Quality for Input / Output values / status (SrcQ_IO)
   // 0 = Good: live, confirmed good;   1 = Good: live, assumed good;
   // 2 = Good: no feedback, assumed good;   8 = Test: Simulated;   9 = Test: Loopback;
   // 10 = Test: Manually Entered;   16 = Uncertain: Live, off-spec;
   // 17 = Uncertain, Substituted at Device / Bus;   18 = Uncertain, Substituted at AOI;
   // 19 = Uncertain, using last known good;    20 = Uncertain, using replacement value;
   // 32 = Bad, Signal Failure;   33 = Bad, Channel Fault;
   // 34 = Bad, Module / Comms Fault;   35 = Bad, Invalid Configuration
   // #####  V3.1-00  2014-06-30:  Added rung for Source/Quality enumerations.  #####
   16: [MOV(1,Wrk_SrcQ) ,XIC(Inp_PVBad) MOV(34,Wrk_SrcQ) ,XIC(Inp_Sim) MOV(10,Wrk_SrcQ) ,MOV(Wrk_SrcQ,SrcQ_IO) ];
   // Source and Quality for primary values / status (SrcQ)
   // 0 = Good: live, confirmed good;   1 = Good: live, assumed good;
   // 2 = Good: no feedback, assumed good;   8 = Test: Simulated;   9 = Test: Loopback;
   // 10 = Test: Manually Entered;   16 = Uncertain: Live, off-spec;
   // 17 = Uncertain, Substituted at Device / Bus;   18 = Uncertain, Substituted at AOI;
   // 19 = Uncertain, using last known good;    20 = Uncertain, using replacement value;
   // 32 = Bad, Signal Failure;   33 = Bad, Channel Fault;
   // 34 = Bad, Module / Comms Fault;   35 = Bad, Invalid Configuration
   // #####  V3.1-00  2014-06-30:  Added rung for Source/Quality enumerations.  #####
   17: [MOV(SrcQ_IO,Wrk_SrcQ) ,XIC(Sts_SubstPV) MOV(18,Wrk_SrcQ) ,MOV(Wrk_SrcQ,SrcQ) ];
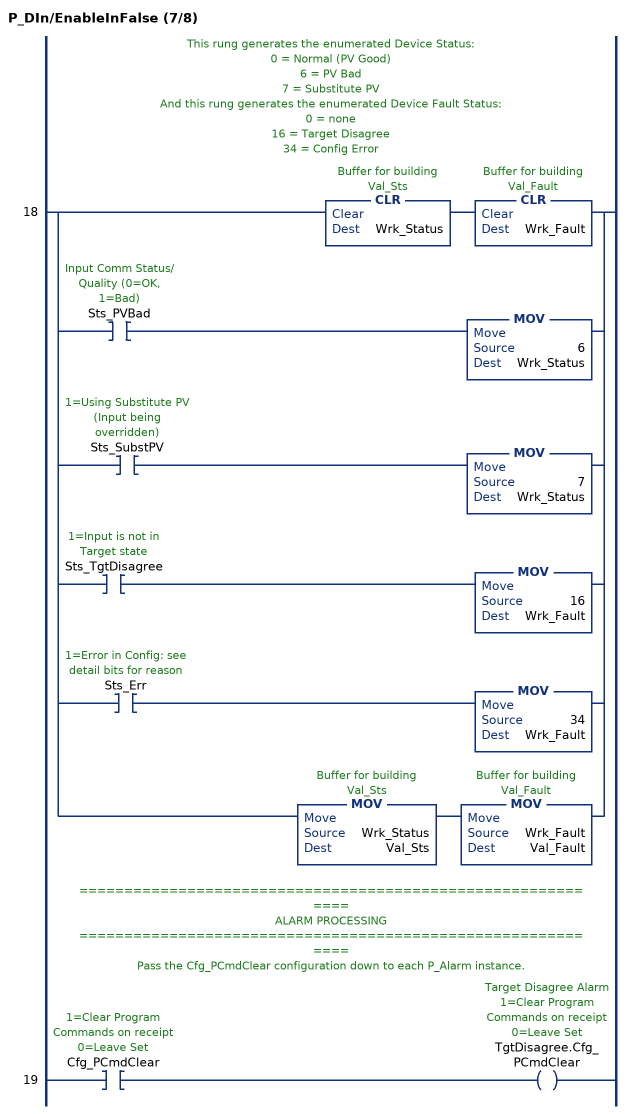
   // This rung generates the enumerated Device Status:
   // 0 = Normal (PV Good)
   // 6 = PV Bad
   // 7 = Substitute PV
   // And this rung generates the enumerated Device Fault Status:
   // 0 = none
   // 16 = Target Disagree
   // 34 = Config Error
   18: [CLR(Wrk_Status) CLR(Wrk_Fault) ,XIC(Sts_PVBad) MOV(6,Wrk_Status) ,XIC(Sts_SubstPV) MOV(7,Wrk_Status) ,XIC(Sts_TgtDisagree) MOV(16,Wrk_Fault) ,XIC(Sts_Err) MOV(34,Wrk_Fault) ,MOV(Wrk_Status,Val_Sts) MOV(Wrk_Fault,Val_Fault) ];
   // ============================================================
   // ALARM PROCESSING
   // ============================================================
   // Pass the Cfg_PCmdClear configuration down to each P_Alarm instance.
   19: XIC(Cfg_PCmdClear)OTE(TgtDisagree.Cfg_PCmdClear);
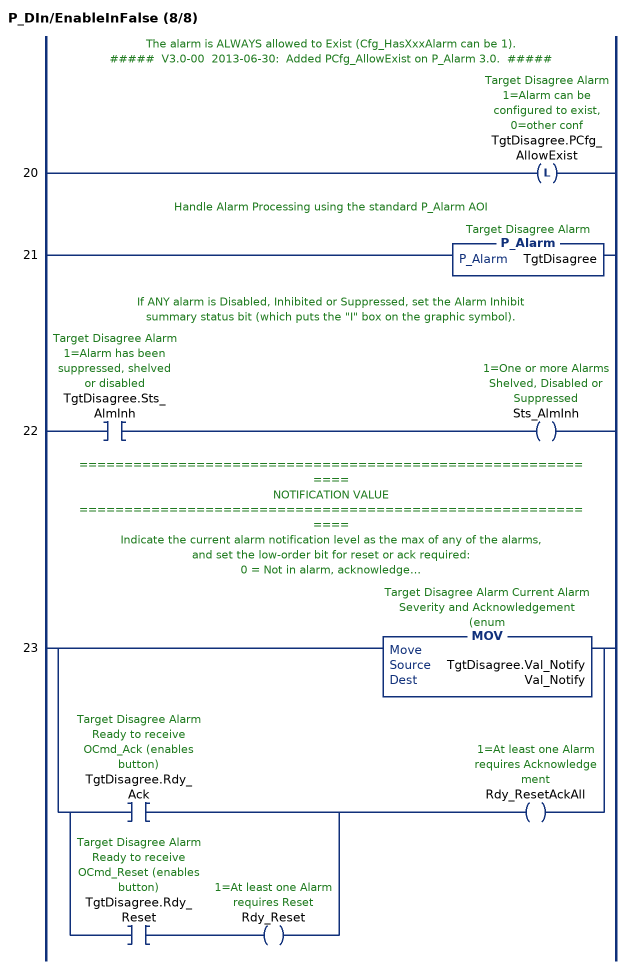
   // The alarm is ALWAYS allowed to Exist (Cfg_HasXxxAlarm can be 1).
   // #####  V3.0-00  2013-06-30:  Added PCfg_AllowExist on P_Alarm 3.0.  #####
   20: OTL(TgtDisagree.PCfg_AllowExist);
   // Handle Alarm Processing using the standard P_Alarm AOI
   21: P_Alarm(TgtDisagree);
   // If ANY alarm is Disabled, Inhibited or Suppressed, set the Alarm Inhibit
   // summary status bit (which puts the "I" box on the graphic symbol).
   22: XIC(TgtDisagree.Sts_AlmInh)OTE(Sts_AlmInh);
   // ============================================================
   // NOTIFICATION VALUE
   // ============================================================
   // Indicate the current alarm notification level as the max of any of the alarms,
   // and set the low-order bit for reset or ack required:
   // 0 = Not in alarm, acknowledged
   // 1 = Not in alarm, unacknowledged or reset required
   // 2 = Low severity alarm, acknowledged
   // 3 = Low severity alarm, unacknowledged
   // 4 = Medium severity alarm, acknowledged
   // 5 = Medium severity alarm, unacknowledged
   // 6 = High severity alarm, acknowledged
   // 7 = High severity alarm, unacknowledged
   // 8 = Urgent severity alarm, acknowledged
   // 9 = Urgent severity alarm, unacknowledged
   // #####  V3.1-00  2014-06-30:  Separated Reset Reqd functions from Val_Notify  #####
   23: [MOV(TgtDisagree.Val_Notify,Val_Notify) ,[XIC(TgtDisagree.Rdy_Ack) ,XIC(TgtDisagree.Rdy_Reset) OTE(Rdy_Reset) ] OTE(Rdy_ResetAckAll) ];
END_ROUTINE
